Staubli VAL3: recursion1.pgx

program recursion1(string x_sString (dimensions=1))
begin
  nNum=nNum+1
  call recursion1(sString)

end
